(* PLC project  *)

CONFIGURATION FSOE_OUT
END_CONFIGURATION
